// TIA Portal V19 export
FUNCTION_BLOCK "VersionCheck"   // FB11, LAD
{ S7_Optimized_Access := 'TRUE' }
// stored: MemoryReserve 100, SetENOAutomatically false
   VAR_INPUT
      CheckVersion : Bool;
   END_VAR
   VAR_OUTPUT
      "Version" : Real;
   END_VAR
   VAR CONSTANT
      CURRENT_VERSION : Real := 0.1;
   END_VAR
BEGIN

REGION Network 1 (SCL)
   IF #CheckVersion THEN
       #Version := #CURRENT_VERSION;
   END_IF;
END_REGION
END_FUNCTION_BLOCK
